Staubli VAL3: USERPAGE.dtx

num keyBoard = 277
public num last = 6
public num nBottomX[2] = 12
num nDelimiterCount
public num nFirst = 2
public num nListHeight[2] = 5
public num nTopX[2] = 20
public num nTopY[2] = 1
num nTxtBoxCol
num nTxtBoxRow
num nTxtBoxWidth
public num nView = 4
num posScroll
public num select = -1
num tpsScroll = 103.137
public string alarm
public string background
public string message
public string nameProject = "false"
public string sItems
public string sTitle = "ItemList"
string sWrkString
public string warning
public bool Show
bool bReadWrite = true
bool bUseEscape
bool bUseRefresh
public bool escape
public bool finish
public bool halt
bool readStr
public bool run
